// TIA Portal project "PLCII_Pro4" (V15.1)

(* hardware
DEVICE "S7-1200 station_1"  S7-1200 Station
   slot 0: "Rack_0"  S7-1200 Rack  Rack  V1.0
   slot 1: "PLC_1"  CPU 1215C DC/DC/Rly  6ES7 215-1HG40-0XB0  V4.2
*)

// ===== PLC "PLC_1"  CPU 1215C DC/DC/Rly =====

VAR_GLOBAL   // PLC tag table "Default tag table"
   "Start" AT %M0.0 : Bool;
   "Sys_runing" AT %M0.1 : Bool;
   "Stop" AT %M0.2 : Bool;
   "Activate" AT %M0.3 : Bool;
   "Sys_Activated" AT %M0.4 : Bool;
END_VAR

DATA_BLOCK "WaterTreatementProcess_DB"   // DB1
{ S7_Optimized_Access := 'TRUE' }
VERSION : 0.1
// stored: InstanceOfName WaterTreatementProcess
"WaterTreatementProcess"
BEGIN
END_DATA_BLOCK

DATA_BLOCK "Sys_variables"   // DB2
{ S7_Optimized_Access := 'TRUE' }
VERSION : 0.1
   VAR
      StartCycle : Bool;
      HomeSW : Bool;
      FillSW : Bool;
      DrainSW : Bool;
      FlushSW : Bool;
      ServoEN : Bool;
      SysState : Int;
      BackToHome : Bool;
      ServoINT : Int;
      CycleCorrectStart : Int;
      Timer_State1 : Time;
      Timer_State2 : Time;
      Timer_State3 : Time;
   END_VAR
BEGIN
END_DATA_BLOCK

DATA_BLOCK "ProcessServoMotor_DB"   // DB3
{ S7_Optimized_Access := 'TRUE' }
VERSION : 0.1
// stored: InstanceOfName ProcessServoMotor
"ProcessServoMotor"
BEGIN
END_DATA_BLOCK

FUNCTION_BLOCK "WaterTreatementProcess"   // FB1, LAD
{ S7_Optimized_Access := 'TRUE' }
VERSION : 0.1
   VAR
      ons1 : Bool;
      ons2 : Bool;
      ons3 : Bool;
      ons4 : Bool;
      ons5 : Bool;
      ons6 : Bool;
      ons7 : Bool;
      ons8 : Bool;
      ons9 : Bool;
      ons10 : Bool;
      ons11 : Bool;
      ons12 : Bool;
      ons13 : Bool;
      ons14 : Bool;
      ons15 : Bool;
   END_VAR
   VAR_TEMP   // added for the SCL form of the ladder/FBD networks
      _w1 : Bool;
      _w2 : Bool;
      _w3 : Bool;
   END_VAR
BEGIN

REGION Network 1
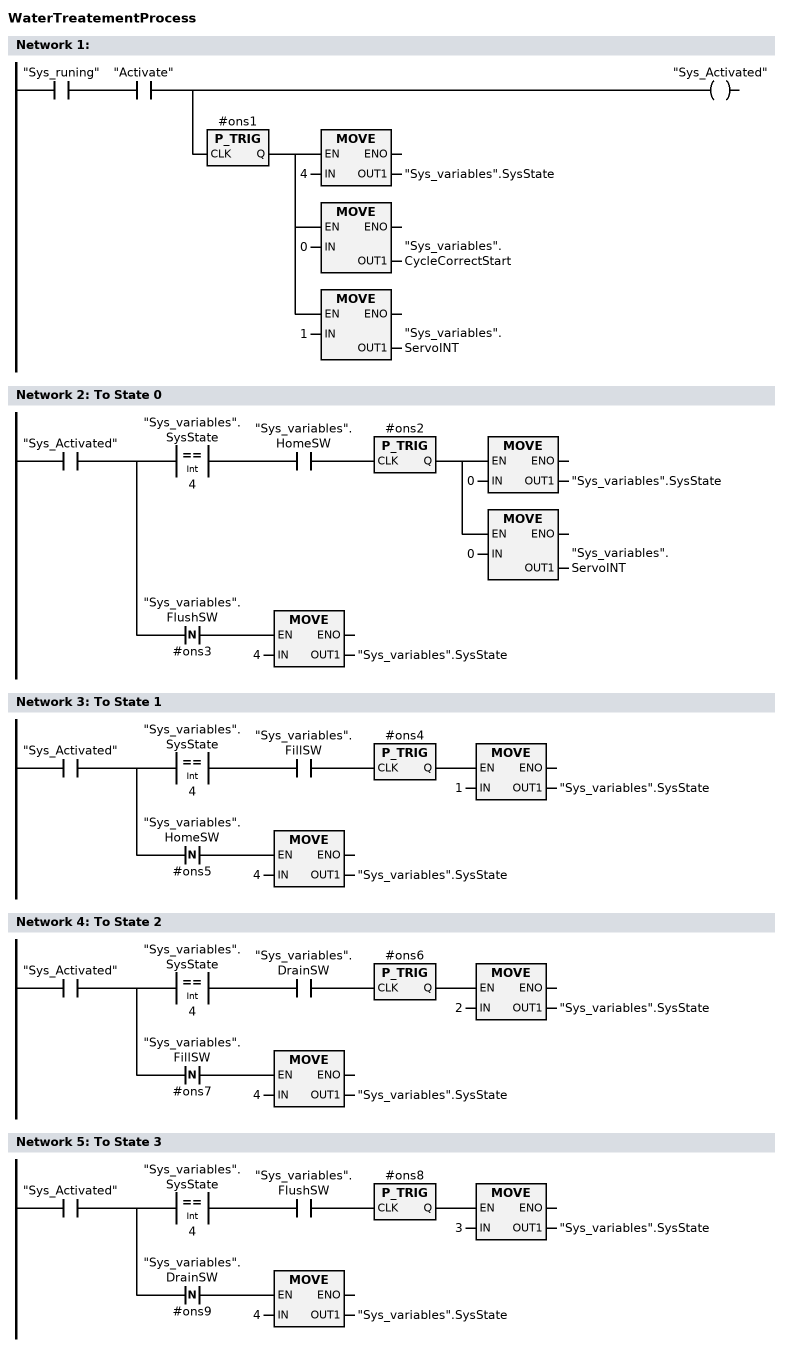
   RUNG wire#powerrail
      Contact( "Sys_runing" )
      Contact( "Activate" )
      wire#w1
      Coil( "Sys_Activated" )
   END_RUNG
   RUNG wire#w1
      P_Trig( #ons1 )
      wire#w2
      Move(in := 4, out1 => "Sys_variables".SysState)
   END_RUNG
   RUNG wire#w2
      Move(in := 0, out1 => "Sys_variables".CycleCorrectStart)
   END_RUNG
   RUNG wire#w2
      Move(in := 1, out1 => "Sys_variables".ServoINT)
   END_RUNG
   // the same network as SCL:
   "Sys_Activated" := "Sys_runing" AND "Activate";
   #_w1 := "Sys_Activated" AND NOT #ons1;   // rising edge
   #ons1 := "Sys_Activated";
   IF #_w1 THEN
       "Sys_variables".SysState := 4;
       "Sys_variables".CycleCorrectStart := 0;
       "Sys_variables".ServoINT := 1;
   END_IF;
END_REGION

REGION Network 2: To State 0
   RUNG wire#powerrail
      Contact( "Sys_Activated" )
      wire#w1
      { S7_Templates := "SrcType := Int" } EQ_Contact(in1 := "Sys_variables".SysState, in2 := 4)
      Contact( "Sys_variables".HomeSW )
      P_Trig( #ons2 )
      wire#w2
      Move(in := 0, out1 => "Sys_variables".SysState)
   END_RUNG
   RUNG wire#w2
      Move(in := 0, out1 => "Sys_variables".ServoINT)
   END_RUNG
   RUNG wire#w1
      N_Contact(operand := "Sys_variables".FlushSW, bit := #ons3)
      Move(in := 4, out1 => "Sys_variables".SysState)
   END_RUNG
   // the same network as SCL:
   #_w1 := "Sys_Activated" AND ("Sys_variables".SysState = 4) AND "Sys_variables".HomeSW;
   #_w2 := #_w1 AND NOT #ons2;   // rising edge
   #ons2 := #_w1;
   IF #_w2 THEN
       "Sys_variables".SysState := 0;
       "Sys_variables".ServoINT := 0;
   END_IF;
   #_w3 := "Sys_Activated" AND NOT "Sys_variables".FlushSW AND #ons3;   // falling edge of "Sys_variables".FlushSW
   #ons3 := "Sys_variables".FlushSW;
   IF #_w3 THEN "Sys_variables".SysState := 4; END_IF;
END_REGION

REGION Network 3: To State 1
   RUNG wire#powerrail
      Contact( "Sys_Activated" )
      wire#w1
      { S7_Templates := "SrcType := Int" } EQ_Contact(in1 := "Sys_variables".SysState, in2 := 4)
      Contact( "Sys_variables".FillSW )
      P_Trig( #ons4 )
      Move(in := 1, out1 => "Sys_variables".SysState)
   END_RUNG
   RUNG wire#w1
      N_Contact(operand := "Sys_variables".HomeSW, bit := #ons5)
      Move(in := 4, out1 => "Sys_variables".SysState)
   END_RUNG
   // the same network as SCL:
   #_w1 := "Sys_Activated" AND ("Sys_variables".SysState = 4) AND "Sys_variables".FillSW;
   #_w2 := #_w1 AND NOT #ons4;   // rising edge
   #ons4 := #_w1;
   IF #_w2 THEN "Sys_variables".SysState := 1; END_IF;
   #_w3 := "Sys_Activated" AND NOT "Sys_variables".HomeSW AND #ons5;   // falling edge of "Sys_variables".HomeSW
   #ons5 := "Sys_variables".HomeSW;
   IF #_w3 THEN "Sys_variables".SysState := 4; END_IF;
END_REGION

REGION Network 4: To State 2
   RUNG wire#powerrail
      Contact( "Sys_Activated" )
      wire#w1
      { S7_Templates := "SrcType := Int" } EQ_Contact(in1 := "Sys_variables".SysState, in2 := 4)
      Contact( "Sys_variables".DrainSW )
      P_Trig( #ons6 )
      Move(in := 2, out1 => "Sys_variables".SysState)
   END_RUNG
   RUNG wire#w1
      N_Contact(operand := "Sys_variables".FillSW, bit := #ons7)
      Move(in := 4, out1 => "Sys_variables".SysState)
   END_RUNG
   // the same network as SCL:
   #_w1 := "Sys_Activated" AND ("Sys_variables".SysState = 4) AND "Sys_variables".DrainSW;
   #_w2 := #_w1 AND NOT #ons6;   // rising edge
   #ons6 := #_w1;
   IF #_w2 THEN "Sys_variables".SysState := 2; END_IF;
   #_w3 := "Sys_Activated" AND NOT "Sys_variables".FillSW AND #ons7;   // falling edge of "Sys_variables".FillSW
   #ons7 := "Sys_variables".FillSW;
   IF #_w3 THEN "Sys_variables".SysState := 4; END_IF;
END_REGION

REGION Network 5: To State 3
   RUNG wire#powerrail
      Contact( "Sys_Activated" )
      wire#w1
      { S7_Templates := "SrcType := Int" } EQ_Contact(in1 := "Sys_variables".SysState, in2 := 4)
      Contact( "Sys_variables".FlushSW )
      P_Trig( #ons8 )
      Move(in := 3, out1 => "Sys_variables".SysState)
   END_RUNG
   RUNG wire#w1
      N_Contact(operand := "Sys_variables".DrainSW, bit := #ons9)
      Move(in := 4, out1 => "Sys_variables".SysState)
   END_RUNG
   // the same network as SCL:
   #_w1 := "Sys_Activated" AND ("Sys_variables".SysState = 4) AND "Sys_variables".FlushSW;
   #_w2 := #_w1 AND NOT #ons8;   // rising edge
   #ons8 := #_w1;
   IF #_w2 THEN "Sys_variables".SysState := 3; END_IF;
   #_w3 := "Sys_Activated" AND NOT "Sys_variables".DrainSW AND #ons9;   // falling edge of "Sys_variables".DrainSW
   #ons9 := "Sys_variables".DrainSW;
   IF #_w3 THEN "Sys_variables".SysState := 4; END_IF;
END_REGION
END_FUNCTION_BLOCK

FUNCTION_BLOCK "ProcessServoMotor"   // FB2, LAD
{ S7_Optimized_Access := 'TRUE' }
VERSION : 0.1
   VAR
      ons1 : Bool;
      ons2 : Bool;
      ons3 : Bool;
      ons4 : Bool;
      ons5 : Bool;
      ons6 : Bool;
      ons7 : Bool;
      ons8 : Bool;
      ons9 : Bool;
      ons10 : Bool;
      StateTimer_State1 : "StateTimer";
      StartTimerSt1 : Bool;
      StartTimerSt2 : Bool;
      StartTimerSt3 : Bool;
   END_VAR
   VAR_TEMP
      varr : Bool;
   END_VAR
   VAR_TEMP   // added for the SCL form of the ladder/FBD networks
      _w1 : Bool;
      _w2 : Bool;
   END_VAR
BEGIN

REGION Network 1
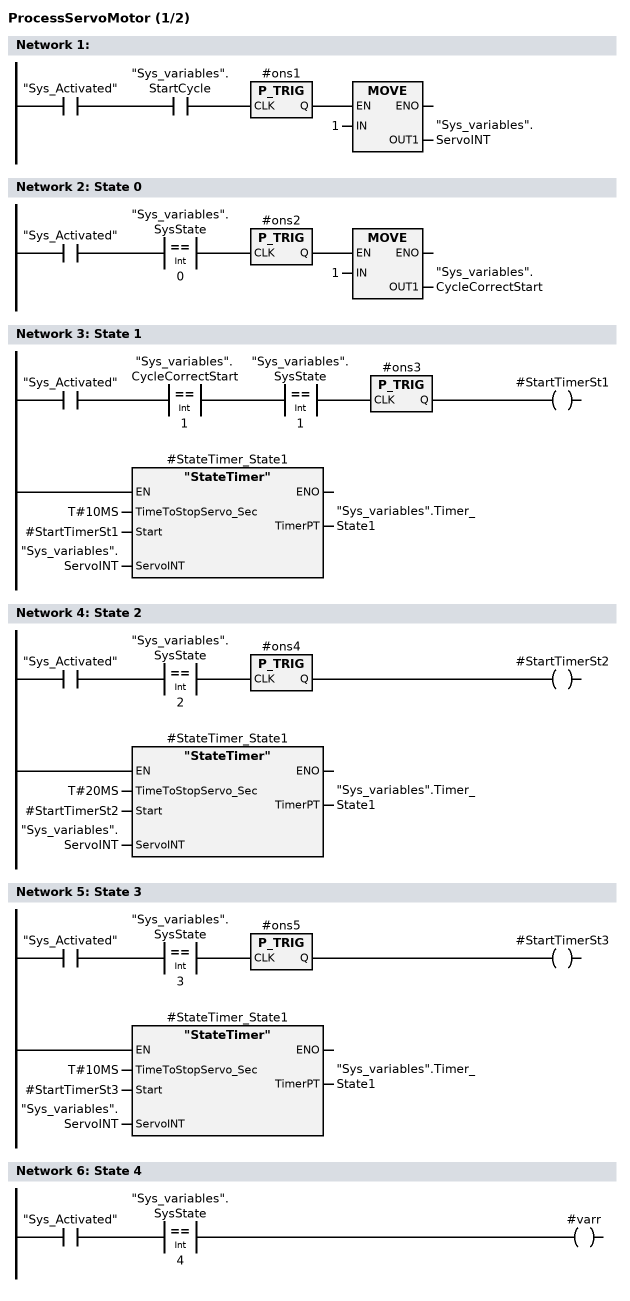
   RUNG wire#powerrail
      Contact( "Sys_Activated" )
      Contact( "Sys_variables".StartCycle )
      P_Trig( #ons1 )
      Move(in := 1, out1 => "Sys_variables".ServoINT)
   END_RUNG
   // the same network as SCL:
   #_w1 := "Sys_Activated" AND "Sys_variables".StartCycle;
   #_w2 := #_w1 AND NOT #ons1;   // rising edge
   #ons1 := #_w1;
   IF #_w2 THEN "Sys_variables".ServoINT := 1; END_IF;
END_REGION

REGION Network 2: State 0
   RUNG wire#powerrail
      Contact( "Sys_Activated" )
      { S7_Templates := "SrcType := Int" } EQ_Contact(in1 := "Sys_variables".SysState, in2 := 0)
      P_Trig( #ons2 )
      Move(in := 1, out1 => "Sys_variables".CycleCorrectStart)
   END_RUNG
   // the same network as SCL:
   #_w1 := "Sys_Activated" AND ("Sys_variables".SysState = 0);
   #_w2 := #_w1 AND NOT #ons2;   // rising edge
   #ons2 := #_w1;
   IF #_w2 THEN "Sys_variables".CycleCorrectStart := 1; END_IF;
END_REGION

REGION Network 3: State 1
   RUNG wire#powerrail
      Contact( "Sys_Activated" )
      { S7_Templates := "SrcType := Int" } EQ_Contact(in1 := "Sys_variables".CycleCorrectStart, in2 := 1)
      { S7_Templates := "SrcType := Int" } EQ_Contact(in1 := "Sys_variables".SysState, in2 := 1)
      P_Trig( #ons3 )
      Coil( #StartTimerSt1 )
   END_RUNG
   RUNG wire#powerrail
      #StateTimer_State1(TimeToStopServo_Sec := T#10MS, Start := #StartTimerSt1, ServoINT := "Sys_variables".ServoINT, TimerPT => "Sys_variables".Timer_State1)
   END_RUNG
   // the same network as SCL:
   #_w1 := "Sys_Activated" AND ("Sys_variables".CycleCorrectStart = 1) AND ("Sys_variables".SysState = 1);
   #_w2 := #_w1 AND NOT #ons3;   // rising edge
   #ons3 := #_w1;
   #StartTimerSt1 := #_w2;
   #StateTimer_State1(TimeToStopServo_Sec := T#10MS,   // "StateTimer"
                      Start := #StartTimerSt1,
                      ServoINT := "Sys_variables".ServoINT,
                      TimerPT => "Sys_variables".Timer_State1);
END_REGION

REGION Network 4: State 2
   RUNG wire#powerrail
      Contact( "Sys_Activated" )
      { S7_Templates := "SrcType := Int" } EQ_Contact(in1 := "Sys_variables".SysState, in2 := 2)
      P_Trig( #ons4 )
      Coil( #StartTimerSt2 )
   END_RUNG
   RUNG wire#powerrail
      #StateTimer_State1(TimeToStopServo_Sec := T#20MS, Start := #StartTimerSt2, ServoINT := "Sys_variables".ServoINT, TimerPT => "Sys_variables".Timer_State1)
   END_RUNG
   // the same network as SCL:
   #_w1 := "Sys_Activated" AND ("Sys_variables".SysState = 2);
   #_w2 := #_w1 AND NOT #ons4;   // rising edge
   #ons4 := #_w1;
   #StartTimerSt2 := #_w2;
   #StateTimer_State1(TimeToStopServo_Sec := T#20MS,   // "StateTimer"
                      Start := #StartTimerSt2,
                      ServoINT := "Sys_variables".ServoINT,
                      TimerPT => "Sys_variables".Timer_State1);
END_REGION

REGION Network 5: State 3
   RUNG wire#powerrail
      Contact( "Sys_Activated" )
      { S7_Templates := "SrcType := Int" } EQ_Contact(in1 := "Sys_variables".SysState, in2 := 3)
      P_Trig( #ons5 )
      Coil( #StartTimerSt3 )
   END_RUNG
   RUNG wire#powerrail
      #StateTimer_State1(TimeToStopServo_Sec := T#10MS, Start := #StartTimerSt3, ServoINT := "Sys_variables".ServoINT, TimerPT => "Sys_variables".Timer_State1)
   END_RUNG
   // the same network as SCL:
   #_w1 := "Sys_Activated" AND ("Sys_variables".SysState = 3);
   #_w2 := #_w1 AND NOT #ons5;   // rising edge
   #ons5 := #_w1;
   #StartTimerSt3 := #_w2;
   #StateTimer_State1(TimeToStopServo_Sec := T#10MS,   // "StateTimer"
                      Start := #StartTimerSt3,
                      ServoINT := "Sys_variables".ServoINT,
                      TimerPT => "Sys_variables".Timer_State1);
END_REGION

REGION Network 6: State 4
   RUNG wire#powerrail
      Contact( "Sys_Activated" )
      { S7_Templates := "SrcType := Int" } EQ_Contact(in1 := "Sys_variables".SysState, in2 := 4)
      Coil( #varr )
   END_RUNG
   // the same network as SCL:
   #varr := "Sys_Activated" AND ("Sys_variables".SysState = 4);
END_REGION

REGION Network 7
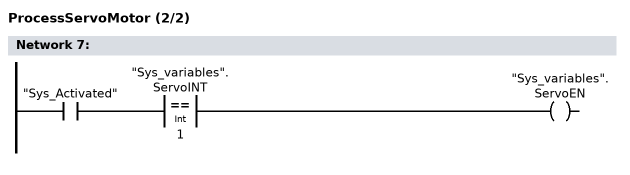
   RUNG wire#powerrail
      Contact( "Sys_Activated" )
      { S7_Templates := "SrcType := Int" } EQ_Contact(in1 := "Sys_variables".ServoINT, in2 := 1)
      Coil( "Sys_variables".ServoEN )
   END_RUNG
   // the same network as SCL:
   "Sys_variables".ServoEN := "Sys_Activated" AND ("Sys_variables".ServoINT = 1);
END_REGION
END_FUNCTION_BLOCK

FUNCTION_BLOCK "StateTimer"   // FB3, LAD
{ S7_Optimized_Access := 'TRUE' }
VERSION : 0.1
   VAR_INPUT
      TimeToStopServo_Sec : Time := T#0s;
      Start : Bool;
   END_VAR
   VAR_OUTPUT
      TimerPT : Time;
   END_VAR
   VAR_IN_OUT
      ServoINT : Int;
   END_VAR
   VAR
      InternTimer : IEC_TIMER;
      BlockActivated : Bool;
      ons1 : Bool;
   END_VAR
   VAR_TEMP
      TimeTempSINT : Int;
      TimeTempMSINT : Int;
      UsedTime : Time;
   END_VAR
   VAR_TEMP   // added for the SCL form of the ladder/FBD networks
      _w1 : Bool;
      _w2 : Bool;
   END_VAR
BEGIN

REGION Network 1
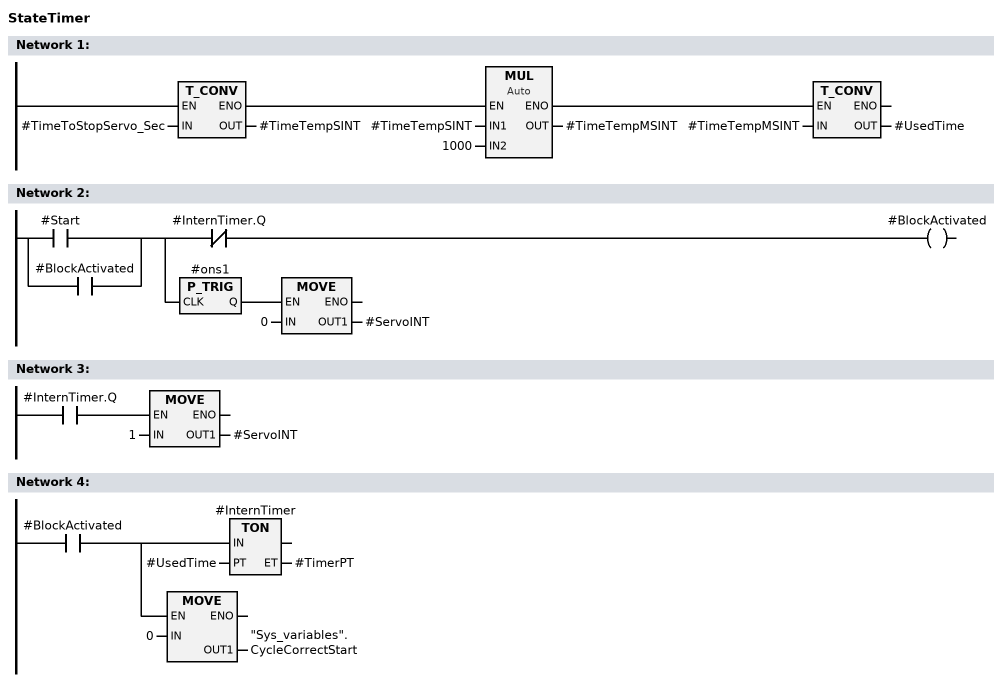
   // ENO of a box is taken as its EN; it also drops when the box reports an error
   #TimeTempSINT := T_CONV(IN := #TimeToStopServo_Sec);
   #TimeTempMSINT := #TimeTempSINT * 1000;
   #UsedTime := T_CONV(IN := #TimeTempMSINT);
END_REGION

REGION Network 2
   RUNG wire#powerrail
      Contact( #Start )
      wire#w1
      I_Contact( #InternTimer.Q )
      Coil( #BlockActivated )
   END_RUNG
   RUNG wire#powerrail
      Contact( #BlockActivated )
   END_RUNG wire#w1
   RUNG wire#w1
      P_Trig( #ons1 )
      Move(in := 0, out1 => #ServoINT)
   END_RUNG
   // the same network as SCL:
   #_w1 := #Start OR #BlockActivated;
   #BlockActivated := #_w1 AND NOT #InternTimer.Q;
   #_w2 := #_w1 AND NOT #ons1;   // rising edge
   #ons1 := #_w1;
   IF #_w2 THEN #ServoINT := 0; END_IF;
END_REGION

REGION Network 3
   RUNG wire#powerrail
      Contact( #InternTimer.Q )
      Move(in := 1, out1 => #ServoINT)
   END_RUNG
   // the same network as SCL:
   IF #InternTimer.Q THEN #ServoINT := 1; END_IF;
END_REGION

REGION Network 4
   #InternTimer.TON(IN := #BlockActivated, PT := #UsedTime, ET => #TimerPT);
   IF #BlockActivated THEN "Sys_variables".CycleCorrectStart := 0; END_IF;
END_REGION
END_FUNCTION_BLOCK

ORGANIZATION_BLOCK "Main"   // OB1, LAD, ProgramCycle
TITLE = "Main Program Sweep (Cycle)"
{ S7_Optimized_Access := 'TRUE' }
VERSION : 0.1
   VAR_INPUT
      Initial_Call : Bool;   // Initial call of this OB
      Remanence : Bool;   // =True, if remanent data are available
   END_VAR
   VAR_TEMP   // added for the SCL form of the ladder/FBD networks
      _w1 : Bool;
   END_VAR
BEGIN

REGION Network 1
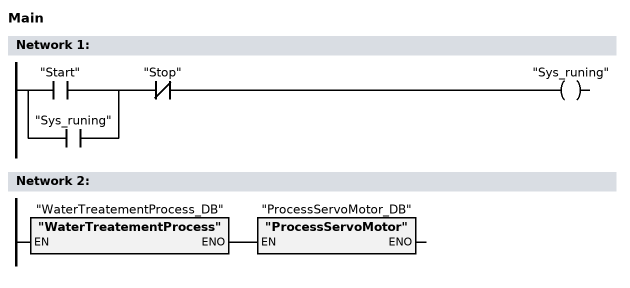
   RUNG wire#powerrail
      Contact( "Start" )
      wire#w1
      I_Contact( "Stop" )
      Coil( "Sys_runing" )
   END_RUNG
   RUNG wire#powerrail
      Contact( "Sys_runing" )
   END_RUNG wire#w1
   // the same network as SCL:
   "Sys_runing" := ("Start" OR "Sys_runing") AND NOT "Stop";
END_REGION

REGION Network 2
   RUNG wire#powerrail
      "WaterTreatementProcess_DB"()
      "ProcessServoMotor_DB"()
   END_RUNG
   // the same network as SCL:
   "WaterTreatementProcess_DB"(ENO => #_w1);   // "WaterTreatementProcess"
   IF #_w1 THEN
       "ProcessServoMotor_DB"();   // "ProcessServoMotor"
   END_IF;
END_REGION
END_ORGANIZATION_BLOCK